# EPICS StreamDevice protocol: protocols/caenels-hs.proto
OutTerminator = CR;
InTerminator = CR;
ReplyTimeout = 2000;
LockTimeout = 10000;

getModel {
    out "VER";
    in "#VER:%s\_%*s";
    @init  {
        out "VER";
        in "#VER:%s\_%*s"
    }
}

getVersion {
    out "VER\r";
    in "%*[^:]:%[^:]:%[^:]:%[^\\r]";
    ExtraInput = Ignore;
}

# getVersion {
#     out "VER";
#     in "#VER:%*s\_%*[^:]:%s";
#     @init {
#         out "VER";
#         in "#VER:%*s\_%*[^:]:%s";
#     };
# }

################################################################################

setEnable {
    out "%{MOFF|MON}";
    in "#AK";
}

setBulkEnable {
    out "%{BOFF|BON}";
    in "#AK";
}

# the commands are MWI (go to setpt without ramp) and MWIR (ramp)
setCurrent {
    out "MWI%(\$1RampEnable){|R}:%f";
    in "#AK";
}

resetStatus {
    out "MRESET";
    in "#AK";
}

################################################################################

getOutputVoltage {
    out "MRV";
    in "#MRV:%f";
}

getOutputCurrent {
    out "MRI";
    in "#MRI:%f" ;
}

getGroundCurrent {
    out "MGC";
    in "#MGC:%f";
}

getDCLinkVoltage {
    out "MRP";
    in "#MRP:%f";
}

getTemperature {
    out "MRT";
    in "#MRT:%f";
}

getStatusMSB {
    out "MST";
    in "#MST:%4x%*4x";
}

getStatusLSB {
    out "MST";
    in "#MST:%*4x%4x";
    @init {
        out "MST";
        in "#MST:%*4x%4x";
    }
}
